(* CoDeSys 2.3.9.41 project: SmarHousePLC110.pro *)
(* Libraries: STANDARD.LIB 4.10.05 11:14:46, IECSFC.LIB 13.4.06 15:51:28, ANALYZATION.LIB 5.10.99 09:05:06 *)

(* PLC configuration (modules and I/O channels)
Fast discrete inputs [I_SIMPLE_INPUT] node 0, in %IB0 out %QB0 {ChannellName = Fast discrete inputs; Filtrationtime = 10000}
  AT %IX0.0 [BitInput] Discrete input 1 {ChannellName = Enter name}
  AT %IX0.1 [BitInput] Discrete input 2 {ChannellName = Enter name}
  AT %IX0.2 [BitInput] Discrete input 3 {ChannellName = Enter name}
  AT %IX0.3 [BitInput] Discrete input 4 {ChannellName = Enter name}
Discrete inputs [ID130] node 1, in %IB1 out %QB1 {ChannellName = Discrete inputs; Filtrationtime_GeneralINP = 10; PinCount = 32}
  REG_INPUT_5_12 AT %IB1.0 [ByteInput] 8 discrete inputs {ChannellName = Enter name}
  REG_INPUT_13_20 AT %IB1.1 [ByteInput] 8 discrete inputs {ChannellName = Enter name}
  REG_INPUT_21_28 AT %IB1.2 [ByteInput] 8 discrete inputs {ChannellName = Enter name}
  REG_INPUT_29_36 AT %IB1.3 [ByteInput] 8 discrete inputs {ChannellName = Enter name}
Fast discrete outputs [OWEN_ID570] node 2, in %IB2 out %QB2 {ChannellName = Fast discrete outputs; SafeValueBool = FALSE; SafeValueBool = FALSE; SafeValueBool = FALSE; SafeValueBool = FALSE; Visibility = No}
  AT %QX2.0 [BitOutput] Fast discrete output 1 {ChannellName = Enter name}
  AT %QX2.1 [BitOutput] Fast discrete output 2 {ChannellName = Enter name}
  AT %QX2.2 [BitOutput] Fast discrete output 3 {ChannellName = Enter name}
  AT %QX2.3 [BitOutput] Fast discrete output 4 {ChannellName = Enter name}
Discrete outputs [ID131] node 3, in %IB3 out %QB3 {ChannellName = Discrete outputs; SafeValueByte = 0; SafeValueByte = 0; SafeValueByteM = 0; PinCount = 24}
  REG_OUT_5_12 AT %QB3.0 [ByteOutput] 8 discrete outputs {ChannellName = Enter name}
  REG_OUT_13_20 AT %QB3.1 [ByteOutput] 8 discrete outputs {ChannellName = Enter name}
  REG_OUT_21_24 AT %QB3.2 [ByteOutput] 4 discrete outputs {ChannellName = Enter name}
AT %IX4.0 [BitInput] Special input {ChannellName = Enter name}
BUZZER AT %QX5.0 [BitOutput] Special output {ChannellName = Enter name}
Modbus [MODBUS_ID302] node 0, in %IB6.0 out %QB6.0 {ChannellName = Modbus}
  TCP [TCP_ID221] node 0, in %IB6.0.0 out %QB6.0.0 {ChannellName = TCP; RemotePort = 502; Visibility = No}
8 bits [8Bit] node 1, in %IB6.1 out %QB6.1 {ChannellName = 8 bit}
  REG_OUT_5_12_FROM_RS AT %QB6.1.0 [ByteOutput] Регистры управления каналами выхода RS {ChannellName = 5-12}
8 bits [8Bit] node 2, in %IB6.2 out %QB6.2 {ChannellName = 8 bit}
  REG_OUT_13_20_FROM_RS AT %QB6.2.0 [ByteOutput] {ChannellName = Enter name}
8 bits [8Bit] node 3, in %IB6.3 out %QB6.3 {ChannellName = 8 bit}
  REG_OUT_21_24_FROM_RS AT %QB6.3.0 [ByteOutput] {ChannellName = Enter name}
8 bits [8Bit] node 4, in %IB6.4 out %QB6.4 {ChannellName = 8 bit}
  AT %QB6.4.0 [ByteOutput] {ChannellName = Enter name}
Float [Float] node 5, in %IB6.5 out %QB6.5 {ChannellName = float}
  EXTERNAL_TEMP_STM_TO_RS AT %QD6.5.0 [FloatOutput] {ChannellName = Enter name}
Float [Float] node 6, in %IB6.6 out %QB6.6 {ChannellName = float}
  INTERNAL_TEMP_STM_TO_RS AT %QD6.6.0 [FloatOutput] {ChannellName = Enter name}
AT %QD7.0 [DWordOutput] Last address {ChannellName = Enter name}
AT %QW7.1 [WordOutput] Last error {ChannellName = Enter name}
RS-485-1 [COM1_USART] node 0, in %IB7.0 out %QB7.0 {ChannellName = RS-485-1; CommunicationSpeed = 57600; Parity = NO PARITY CHECK; BitLength = 8 bits; StopLength = One stop bit; InterfaceType = RS485; FrameOriented = RTU; Timeout = 1000; Visibility = No}
AT %QB7.1.0 [ComChannel] Command (0xff - Start) {ChannellName = Enter name}
INTERNAL_TEMP_STM AT %QD7.1.0.0 [FloatOutput] {ChannellName = Enter name}
EXTERNAL_TEMP_STM AT %QD7.1.1.0 [FloatOutput] {ChannellName = Enter name}
*)

(* POU PLC_PRG, ST *)
PROGRAM PLC_PRG
VAR
	PLC_INIT_FLAG:BOOL:=FALSE;



	OUT6_IN6_CHECK_AND_TOOGLE:  CHECK_INPUT_TOOGLE_OUT;
	OUT5_IN5_CHECK_AND_TOOGLE:  CHECK_INPUT_TOOGLE_OUT;
	OUT6_IN5_CHECK_AND_TOOGLE:  CHECK_INPUT_TOOGLE_OUT;

	IN6_ALL_LIGHT_OFF_CHECK:	CHECK_INPUT_PRESS_MS;
	IN6_ALL_FLOR_OFF_CHECK:	CHECK_INPUT_PRESS_MS;

	ALL_LIGHT_OFF_FLAG:BOOL:=FALSE;
	ALL_FLOR_OFF_FLAG:BOOL:=FALSE;

END_VAR
IF PLC_INIT_FLAG = FALSE THEN (* инициализация переменных *)
	PLC_INIT_FLAG:= TRUE;
	REG_OUT_5_12_FROM_RS:=0;
 	REG_OUT_13_20_FROM_RS:=0;
 	REG_OUT_21_24_FROM_RS:=0;

	OUT6_IN6_CHECK_AND_TOOGLE(INIT_OUTPUT_CHANNEL:=6, INIT_INPUT_CAHANNEL:=6);(*определение функциональных блоков НАЖАТИЕ*)
	OUT6_IN5_CHECK_AND_TOOGLE(INIT_OUTPUT_CHANNEL:=6, INIT_INPUT_CAHANNEL:=5);
	OUT5_IN5_CHECK_AND_TOOGLE(INIT_OUTPUT_CHANNEL:=5, INIT_INPUT_CAHANNEL:=5);

	IN6_ALL_LIGHT_OFF_CHECK(INIT_INPUT_CAHANNEL:=6, INIT_TIME_MS := 3000);(*определение функционального блока УДЕРЖАНИЕ*)
	IN6_ALL_FLOR_OFF_CHECK(INIT_INPUT_CAHANNEL:=6, INIT_TIME_MS := 5000);

(*	WriteOUTPUT(20,TRUE);
	WriteOUTPUT(19,TRUE); *)
	SET_ENERGY_FLAG(TRUE);


END_IF








(*

REG_OUT_5_12
REG_OUT_13_20 - Регистры выходов ПЛК  (1<<0) = 5 , (1<<0) = 13
 осталось 1-4 фаст выходы и 20 -24 доп обычные выходы 

REG_INPUT_5_12 - входы
REG_INPUT_13_20
REG_INPUT_21_28
REG_INPUT_29_36

*)


(*   прежде чем что то переключить применим выходы из Home Assistance  *)
	REG_OUT_5_12	 := REG_OUT_5_12_FROM_RS;
	REG_OUT_13_20 := REG_OUT_13_20_FROM_RS;
	REG_OUT_21_24:=  REG_OUT_21_24_FROM_RS;
	EXTERNAL_TEMP_STM_TO_RS := EXTERNAL_TEMP_STM;
	INTERNAL_TEMP_STM_TO_RS  := INTERNAL_TEMP_STM;

(*  переключение каналов по клику  *)
	OUT6_IN6_CHECK_AND_TOOGLE();
	OUT5_IN5_CHECK_AND_TOOGLE();

(*  переключение каналов по удержанию  *)
	IN6_ALL_LIGHT_OFF_CHECK( EVENT => ALL_LIGHT_OFF_FLAG );
	IF ALL_LIGHT_OFF_FLAG = TRUE THEN(*мастер выключатель*)

		WriteOUTPUT(5,FALSE);
		WriteOUTPUT(6,FALSE);
		WriteOUTPUT(7,FALSE);
		WriteOUTPUT(8,FALSE);
		WriteOUTPUT(9,FALSE);
		WriteOUTPUT(10,FALSE);
		WriteOUTPUT(11,FALSE);
		WriteOUTPUT(12,FALSE);
		WriteOUTPUT(13,FALSE);
		WriteOUTPUT(14,FALSE);
		WriteOUTPUT(15,FALSE);
	END_IF

	IN6_ALL_FLOR_OFF_CHECK( EVENT => ALL_FLOR_OFF_FLAG );
	IF ALL_FLOR_OFF_FLAG = TRUE THEN(*мастер выключатель*)
		SET_ENERGY_FLAG(FALSE);
		WriteOUTPUT(5,FALSE);
		WriteOUTPUT(6,FALSE);
		WriteOUTPUT(7,FALSE);
		WriteOUTPUT(8,FALSE);
		WriteOUTPUT(9,FALSE);
		WriteOUTPUT(10,FALSE);
		WriteOUTPUT(11,FALSE);
		WriteOUTPUT(12,FALSE);
		WriteOUTPUT(13,FALSE);
		WriteOUTPUT(14,FALSE);
		WriteOUTPUT(15,FALSE);

		WriteOUTPUT(20,FALSE);
	END_IF


TEST_KEY := REG_INPUT_29_36.7;
END_PROGRAM

(* POU CHECK_INPUT_TOOGLE_OUT, ST *)
FUNCTION_BLOCK CHECK_INPUT_TOOGLE_OUT
VAR_INPUT
	INIT_INPUT_CAHANNEL: BYTE:=0;
	INIT_OUTPUT_CHANNEL: BYTE:=0;
END_VAR
VAR_OUTPUT
END_VAR
VAR
	OUTPUT_CHANNEL: BYTE:=0;
	INPUT_CAHANNEL: BYTE:=0;
	FLAG: BOOL;
	CHANNEL_OUTPUT_BIT  : DWORD;
	INPUT_REG_CURRENT_DATA: BYTE;
END_VAR
IF OUTPUT_CHANNEL = 0 OR INPUT_CAHANNEL=0  THEN(*ПРОВЕРКА КОРРЕКТНОСТИ И ИНИЦАЛИЗАЦИИ*)
	IF OUTPUT_CHANNEL = 0 AND  INIT_OUTPUT_CHANNEL <> 0 THEN
		OUTPUT_CHANNEL := INIT_OUTPUT_CHANNEL;
	END_IF

	IF INPUT_CAHANNEL = 0 AND  INIT_INPUT_CAHANNEL <> 0 THEN
		INPUT_CAHANNEL := INIT_INPUT_CAHANNEL;
	END_IF

	RETURN;
END_IF

(*инициализация выходного КАНАЛА ПРИ OUTPUT_CHANNEL == 255 *)

IF  CheckINPUT(INPUT_CAHANNEL) =  TRUE AND FLAG = FALSE THEN
		ToogleOUTPUT(OUTPUT_CHANNEL) ;
		FLAG := TRUE;
	ELSE
		IF  CheckINPUT(INPUT_CAHANNEL) =  FALSE AND FLAG = TRUE THEN
			FLAG := FALSE;
		END_IF
END_IF
END_FUNCTION_BLOCK

(* POU CheckINPUT, ST *)
FUNCTION CheckINPUT : BOOL
VAR_INPUT
	INPUT_CAHANNEL: BYTE;
END_VAR
VAR
	CHANNEL_INPUT_BIT : BYTE;
	INPUT_REG_CURRENT_DATA:BYTE;
END_VAR
CASE INPUT_CAHANNEL OF
		5..12:
			CHANNEL_INPUT_BIT := INPUT_CAHANNEL - 5;
			INPUT_REG_CURRENT_DATA := REG_INPUT_5_12;
		13..20:
			CHANNEL_INPUT_BIT := INPUT_CAHANNEL - 13;
			INPUT_REG_CURRENT_DATA := REG_INPUT_13_20;
		21..28:
			CHANNEL_INPUT_BIT := INPUT_CAHANNEL - 21;
			INPUT_REG_CURRENT_DATA := REG_INPUT_21_28;
		29..36:
			CHANNEL_INPUT_BIT := INPUT_CAHANNEL - 29;
			INPUT_REG_CURRENT_DATA := REG_INPUT_29_36;
		ELSE
			CheckINPUT:= FALSE;
			RETURN;
END_CASE

IF  ( INPUT_REG_CURRENT_DATA  AND SHL(1,CHANNEL_INPUT_BIT)  ) = SHL(1,CHANNEL_INPUT_BIT)   THEN
	CheckINPUT:=  TRUE;
ELSE
	CheckINPUT:= FALSE;
END_IF
END_FUNCTION

(* POU ToogleOUTPUT, ST *)
FUNCTION ToogleOUTPUT : BOOL
VAR_INPUT
	OUTPUT_CHANNEL:BYTE;
END_VAR
VAR

END_VAR
IF CheckOUTPUT(OUTPUT_CHANNEL) = TRUE THEN
	WriteOUTPUT(OUTPUT_CHANNEL,FALSE);
ELSE
	WriteOUTPUT(OUTPUT_CHANNEL,TRUE);
END_IF
END_FUNCTION

(* POU CheckOUTPUT, ST *)
FUNCTION CheckOUTPUT : BOOL
VAR_INPUT
	OUTPUT_CHANNEL: BYTE;
END_VAR
VAR
	CHANNEL_OUTPUT_BIT:BYTE;
	OUT_REG_CARRENT_DATA:BYTE;
END_VAR
CASE OUTPUT_CHANNEL OF
		5..12:
			CHANNEL_OUTPUT_BIT := OUTPUT_CHANNEL - 5;
			OUT_REG_CARRENT_DATA  := REG_OUT_5_12;

		13..20:
			CHANNEL_OUTPUT_BIT := OUTPUT_CHANNEL - 13;
			OUT_REG_CARRENT_DATA  := REG_OUT_13_20 ;

		21..24:
			CHANNEL_OUTPUT_BIT := OUTPUT_CHANNEL - 21;
			OUT_REG_CARRENT_DATA := REG_OUT_21_24 ;
END_CASE

IF (OUT_REG_CARRENT_DATA  AND  SHL(1 , CHANNEL_OUTPUT_BIT) )  =  SHL(1 , CHANNEL_OUTPUT_BIT)  THEN
	CheckOUTPUT := TRUE;
ELSE
	CheckOUTPUT := FALSE;
END_IF

(*


IF (OUT_REG_CARRENT_DATA  AND  SHL(1 , CHANNEL_OUTPUT_BIT) )  =  SHL(1 , CHANNEL_OUTPUT_BIT)  THEN
     *)
END_FUNCTION

(* POU WriteOUTPUT, ST *)
FUNCTION WriteOUTPUT : BOOL
VAR_INPUT
	OUTPUT_CHANNEL: BYTE;
	OUTPUT_STATE:BOOL;
END_VAR
VAR
	CHANNEL_OUTPUT_BIT:BYTE;
END_VAR
IF OUTPUT_STATE = TRUE THEN

		CASE OUTPUT_CHANNEL OF
				5..12:
					CHANNEL_OUTPUT_BIT := OUTPUT_CHANNEL - 5;
					REG_OUT_5_12 := REG_OUT_5_12  OR SHL(1 , CHANNEL_OUTPUT_BIT) ;
				13..20:
					CHANNEL_OUTPUT_BIT := OUTPUT_CHANNEL - 13;
					REG_OUT_13_20 := REG_OUT_13_20  OR SHL(1 , CHANNEL_OUTPUT_BIT) ;
				21..24:
					CHANNEL_OUTPUT_BIT := OUTPUT_CHANNEL - 21;
					REG_OUT_21_24 := REG_OUT_21_24  OR SHL(1 , CHANNEL_OUTPUT_BIT) ;
				ELSE
					RETURN;
		END_CASE
		SET_ENERGY_FLAG(TRUE);(*ПРИ АКТИВАЦИИ КАНАЛА ВКЛЮЧЕМ МАСТЕР*)

ELSE

		CASE OUTPUT_CHANNEL OF
				5..12:
					CHANNEL_OUTPUT_BIT := OUTPUT_CHANNEL - 5;
					REG_OUT_5_12 := REG_OUT_5_12  AND NOT SHL(1 , CHANNEL_OUTPUT_BIT) ;
				13..20:
					CHANNEL_OUTPUT_BIT := OUTPUT_CHANNEL - 13;
					REG_OUT_13_20 := REG_OUT_13_20  AND NOT SHL(1 , CHANNEL_OUTPUT_BIT) ;
				21..24:
					CHANNEL_OUTPUT_BIT := OUTPUT_CHANNEL - 21;
					REG_OUT_21_24 := REG_OUT_21_24  AND NOT SHL(1 , CHANNEL_OUTPUT_BIT) ;
				ELSE
					RETURN;
		END_CASE
END_IF

SaveCarrentOutStateForRS();
END_FUNCTION

(* POU SET_ENERGY_FLAG, ST *)
FUNCTION SET_ENERGY_FLAG : BOOL
VAR_INPUT
	ENABLE_FLAG:BOOL:=FALSE;
END_VAR
VAR
	MASTER_OUTPUT: BYTE:=24; (*МАСТЕР ВЫХОД*)

END_VAR
MASTER_OUTPUT:=24;
IF ENABLE_FLAG = TRUE THEN

CASE MASTER_OUTPUT OF
				5..12:
					REG_OUT_5_12 := REG_OUT_5_12  OR SHL(1 , MASTER_OUTPUT - 5) ;
				13..20:
					REG_OUT_13_20 := REG_OUT_13_20  OR SHL(1 , MASTER_OUTPUT - 13) ;
				21..24:
					REG_OUT_21_24 := REG_OUT_21_24  OR SHL(1 , MASTER_OUTPUT - 21) ;
				ELSE
					RETURN;
		END_CASE

ELSE
		CASE MASTER_OUTPUT OF
				5..12:
					REG_OUT_5_12 := REG_OUT_5_12  AND NOT SHL(1 ,  MASTER_OUTPUT - 5) ;
				13..20:
					REG_OUT_13_20 := REG_OUT_13_20  AND NOT SHL(1 , MASTER_OUTPUT - 13) ;
				21..24:
					REG_OUT_21_24 := REG_OUT_21_24  AND NOT SHL(1 , MASTER_OUTPUT - 21) ;
				ELSE
					RETURN;
		END_CASE
END_IF

SaveCarrentOutStateForRS();
END_FUNCTION

(* POU SaveCarrentOutStateForRS, ST *)
FUNCTION SaveCarrentOutStateForRS : BOOL
VAR_INPUT

END_VAR
VAR
END_VAR
	REG_OUT_5_12_FROM_RS 	:= REG_OUT_5_12;
	REG_OUT_13_20_FROM_RS	:= REG_OUT_13_20 ;
	REG_OUT_21_24_FROM_RS	:= REG_OUT_21_24 ;
END_FUNCTION

(* POU CHECK_INPUT_PRESS_MS, ST *)
FUNCTION_BLOCK CHECK_INPUT_PRESS_MS
VAR_INPUT
	INIT_INPUT_CAHANNEL: BYTE:=0;
	INIT_TIME_MS:UINT:=0;
END_VAR
VAR_OUTPUT
	EVENT:BOOL:=FALSE;
END_VAR
VAR

	INPUT_CAHANNEL: BYTE:=0;
	TIME_MS:UINT :=0;
	COUNTER_MS:UINT :=0;
	FLAG:BOOL:=FALSE;
END_VAR
IF  INPUT_CAHANNEL=0  OR TIME_MS = 0 THEN(*ПРОВЕРКА КОРРЕКТНОСТИ И ИНИЦАЛИЗАЦИИ*)
	IF TIME_MS = 0 AND  INIT_TIME_MS <> 0 THEN
		TIME_MS := INIT_TIME_MS;
	END_IF

	IF INPUT_CAHANNEL = 0 AND  INIT_INPUT_CAHANNEL <> 0 THEN
		INPUT_CAHANNEL := INIT_INPUT_CAHANNEL;
	END_IF

	RETURN;
END_IF


IF  CheckINPUT(INPUT_CAHANNEL) =  TRUE AND FLAG= FALSE THEN
		COUNTER_MS:= COUNTER_MS+1;


		IF(TIME_MS = 5000) THEN
			IF COUNTER_MS >= 3500 THEN
				BUZZER:=TRUE;
			END_IF
		END_IF

		IF COUNTER_MS >= TIME_MS THEN
			COUNTER_MS := 0;
			EVENT:= TRUE;
			FLAG:= TRUE;
		END_IF
	ELSE
		COUNTER_MS:=0;
		EVENT:= FALSE;
		IF(TIME_MS = 5000) THEN
			BUZZER:=FALSE;
		END_IF
		IF  CheckINPUT(INPUT_CAHANNEL) =  FALSE AND FLAG= TRUE THEN
			 FLAG := FALSE;
		END_IF
END_IF
END_FUNCTION_BLOCK
